PROGRAM MAIN
VAR
END_VAR

END_PROGRAM

(* stored: Version 1.1.0.1
   POU MAIN: Id {7d0d81e4-aaff-4a57-ba86-23f249594456} *)
